FUNCTION_BLOCK EL3052
VAR
	_io : EL3xx2_Data;
	{attribute addProperty Name "WcState"}
	_wcState : WcStateInputToggle;
	{attribute addProperty Name "Info data"}
	_infoData : InfoDataAds;
END_VAR

PROPERTY IO : REFERENCE TO EL3xx2_Data
GET
IO REF= _io;
END_GET
END_PROPERTY

PROPERTY WcState : REFERENCE TO WcStateInputToggle
GET
WcState REF= _wcState;
END_GET
END_PROPERTY

END_FUNCTION_BLOCK

(* stored: Version 1.1.0.1, ProductVersion 3.1.4024.9
   POU EL3052: Id {637cddb0-6704-0547-0d01-1a2cbadbc2e5}, SpecialFunc None
   Property IO: Id {b5bd322f-fd8d-090f-16a9-cda476cd8d46}
   Get Get: Id {d5515295-fd0d-0fac-3e5a-df4fc93caf53}
   Property WcState: Id {a178a0d6-908d-0881-3379-a82e89882f31}
   Get Get: Id {53660da9-bf1c-05fe-00e6-d10032705c81} *)
